{attribute 'no_explicit_call' := 'Do not call the body - Stick to OOP'}
FUNCTION_BLOCK FB_EtherCAT_Trigger EXTENDS FB_CameraController_Base IMPLEMENTS I_SwTimestamp_Mode
VAR
	nStartTime 				AT %Q*	: T_DCTIME64;			// Trigger time stamp
	nActivate				AT %Q*	: USINT; 				// 0 -> 3 use new time in terminal
	
	{attribute 'hide'}
	nTriggerDelay 			: UDINT := 0;					// The given trigger time is delayed by this value. E.g. to wait for the maximum lighting value before taking a picture  [in 100ns]
	
	{attribute 'hide'}
	eState					: E_StateTerminal;				// Current terminal state
END_VAR

{attribute 'monitoring' := 'call'}
//Module already has a task - already a trigger active
PROPERTY Busy : BOOL
GET
Busy := (THIS^.eState = E_StateTerminal.TRIGGERING) OR (THIS^.eState = E_StateTerminal.RESETING) OR (THIS^.eState = E_StateTerminal.RESET);
END_GET
END_PROPERTY

{attribute 'monitoring' := 'call'}
PROPERTY Operational : BOOL
GET
Operational := (THIS^.eState = E_StateTerminal.READY) OR (THIS^.eState = E_StateTerminal.TRIGGERING);
END_GET
END_PROPERTY

METHOD PUBLIC Reset : HRESULT
VAR_INPUT
END_VAR
IF THIS^.eState = E_StateTerminal.ERROR THEN
	fbFeedback.ActiveCommand := 'Reset';
	fbFeedback.Busy := TRUE;	

	THIS^.eState := E_StateTerminal.RESET;
END_IF
END_METHOD

{attribute 'monitoring' := 'call'}
PROPERTY PUBLIC State : E_StateTerminal
GET
State := THIS^.eState;
END_GET
END_PROPERTY

METHOD PUBLIC Trigger : HRESULT
VAR_INPUT
	//The data type T_DCTIME64 represents the distributed clock system time (abbreviated as DC time) as a linear 64-bit integer value. 
	//The time is expressed in nanoseconds since 1/1/2000 UTC. The smallest unit is a nanosecond.
	//F_GetCurDcTickTime64()
	nDCTimeStamp	: T_DCTIME64;
END_VAR
(* Check if the trigger is minimum 3 EtherCat cycles in future *)
IF (nDCTimeStamp + THIS^.nTriggerDelay) < THIS^.NextPossibleTriggerTime THEN
	Trigger := E_FAIL;
	RETURN;
END_IF

(* Check if not in wrong state *)
IF NOT (THIS^.eState = E_StateTerminal.READY) THEN
	Trigger := E_FAIL;
	RETURN;
END_IF

fbFeedback.ActiveCommand := 'Trigger';
fbFeedback.Busy := TRUE;	


THIS^.nStartTime := nDCTimeStamp + THIS^.nTriggerDelay;
THIS^.nActivate := 3; (*Activate*)

THIS^.eState := E_StateTerminal.TRIGGERING;
Trigger := S_OK;
END_METHOD

{attribute 'monitoring' := 'call'}
// The given trigger time is delayed by this value. E.g. to wait for the maximum lighting value before taking a picture  [in 1ns]
PROPERTY TriggerDelay_1ns : UDINT
GET
TriggerDelay_1ns := THIS^.nTriggerDelay;
END_GET
SET
THIS^.nTriggerDelay := TriggerDelay_1ns;
END_SET
END_PROPERTY

METHOD PUBLIC Update : HRESULT
VAR_INST
	{attribute 'hide'}
	fbTimeout : TON;
END_VAR
(* Handle terminal state machine *)
CASE THIS^.eState OF
	(* Reset all control variables *)
	E_StateTerminal.RESET:
		//THIS^.bReset := TRUE;
		THIS^.eState := E_StateTerminal.RESETING;
		
	(* Reset all control variables *)
	E_StateTerminal.RESETING:
		//THIS^.bReset := FALSE;
		THIS^.eState := E_StateTerminal.INIT;	
		
	(* Enable terminal if ready *)
	E_StateTerminal.INIT:			
		THIS^.eState := E_StateTerminal.READY;

	(* Terminal is ready *)
	E_StateTerminal.READY:
		fbFeedback.Done := TRUE;
		THIS^.nActivate := 0;
		
		
	(* Terminal is triggering *)
	E_StateTerminal.TRIGGERING:
		//WaitForTriggerDone:
		IF (F_GetCurDcTaskTime64()(*1ns*) >= (THIS^.nStartTime)) THEN
			//Befor leave triggering, stay 1 cycle in Activate=0
			IF THIS^.nActivate = 0 THEN
				THIS^.eState := E_StateTerminal.READY;
			ELSE 
				THIS^.nActivate := 0;(*Deactivate*)
			END_IF

		 END_IF
			
	
	(* Error occured *)	
	E_StateTerminal.ERROR:
		fbFeedback.HR := E_FAIL;
		IF NOT THIS^.fbAlarmGeneral.bRaised THEN
			THIS^.fbAlarmGeneral.Raise(0);	
		END_IF
		
		IF (THIS^.fbAlarmGeneral.eConfirmationState = TcEventConfirmationState.Confirmed) THEN
			THIS^.Reset();			
		END_IF			
END_CASE

(* Timeout if an actingstate is to long active *)
fbTimeout.IN := (THIS^.eState = E_StateTerminal.INIT) OR (THIS^.eState = E_StateTerminal.RESETING) OR (THIS^.eState = E_StateTerminal.TRIGGERING);
fbTimeout.PT := T#5S;
fbTimeout();
IF fbTimeout.Q THEN
	THIS^.eState := E_StateTerminal.ERROR;
END_IF
END_METHOD

END_FUNCTION_BLOCK

(* stored: Version 1.1.0.1, ProductVersion 3.1.4024.12
   POU FB_EtherCAT_Trigger: Id {d2cacf00-fad4-437b-81ab-be54172ac98a}, SpecialFunc None
   Property Busy: Id {11d9b0fe-062e-4831-ac97-647831f44ea6}
   Get Get: Id {55eeb9f5-3d99-4c76-80b3-143d6f87db8f}
   Property Operational: Id {4c68750d-8963-4b4b-92df-834ea445e3e7}
   Get Get: Id {e79018bc-f0dd-4892-997e-9c950bfa4415}
   Method Reset: Id {aebbfcaa-e4d5-4af1-9340-320438fac784}
   Property State: Id {28c5230e-3ca2-4a09-b82f-5ab144706d9d}
   Get Get: Id {5529493e-2637-4e81-b25c-3351bb767e07}
   Method Trigger: Id {01fddff3-ea8e-4eb3-9b19-060134a068a7}
   Property TriggerDelay_1ns: Id {8db5f746-f1d6-477d-95ab-c5bd2335534b}
   Get Get: Id {8b18f878-24e8-4c4e-8688-2847169a3bcd}
   Set Set: Id {e741103f-7048-4e99-860e-ae936535d08b}
   Method Update: Id {66b4d5b0-85ea-4970-aa32-d8ac55831f0c} *)
